{attribute 'GeneratedUsingTerminal: EL6690-0002-0000'}
{attribute addProperty BoxType "EL6690-0002-0000"}
{attribute addProperty Id "CycleTimerAT %I*ARRAY [0..2] OF USINT0ErrorCodeAT %I*BYTE1"}
{attribute addProperty CRC "3540894527"}
{attribute addProperty Size "1"}
TYPE Status_D30DC33F :
STRUCT
	{attribute addProperty Name "CycleTimer"}
	CycleTimer AT %I* : ARRAY [0..2] OF USINT;
	{attribute addProperty Name "ErrorCode"}
	ErrorCode AT %I* : BYTE;
END_STRUCT
END_TYPE

(* stored: Version 1.2.0.0, ProductVersion 3.1.4024.9
   DUT Status_D30DC33F: Id {5ea4be67-c254-4b19-8973-94c9afc38d7b} *)
